# B&R Automation Studio project TestOpenpowerlink
Automation Studio 4.3.11.134 SP

## Configuration Config1

CPU X20CP3586, AutomationRuntime N4.34, Build 4.1.2, Vc V4.34.3

### Task classes (Cpu.sw)
```
Cyclic#4:
  Program <- Program.prg
Libraries: AsIOAcc, runtime, BLLibrarys
```

### Hardware
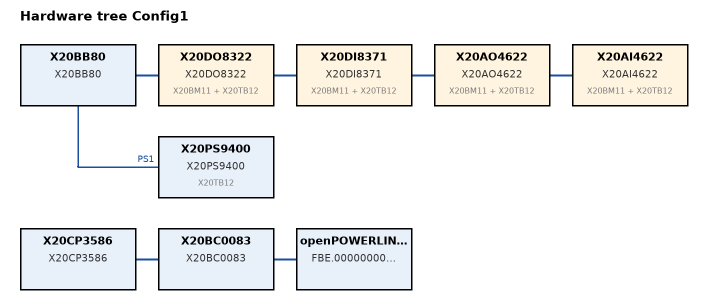
```
X20AI4622 : X20AI4622 v1.0.4.0  [SS1 -> X20TB12d.SS; SL -> X20BM11c.SL1]
  Supervision = off
  LowerLimit = -8192
  ChannelType01 = 4 to 20mA
  ChannelType02 = 4 to 20mA
  ChannelType03 = 4 to 20mA
  ChannelType04 = 4 to 20mA
X20AO4622 : X20AO4622 v1.2.0.0  [SS1 -> X20TB12c.SS; SL -> X20BM11b.SL1]
  Supervision = off
  ChannelType01 = 4 to 20mA
  ChannelType02 = 4 to 20mA
  ChannelType03 = 4 to 20mA
  ChannelType04 = 4 to 20mA
X20BB80 : X20BB80 v1.0.2.0
X20BC0083 : X20BC0083 v2.11.1.0  [PLK1 -> X20CP3586.IF3 (NodeNumber=2) [Cable Type=PowerlinkCable, Length=10, Version=1.0.0.1]; PLK2 -> openPOWERLINK_device.PLK1 (NodeNumber=2) [Cable Type=PowerlinkCable, Length=10, Version=1.0.0.1]; SL -> X20BB80.SL1]
  Supervision = off
X20BM11 : X20BM11 v1.0.0.1  [X2X1 -> X20BB80.IF1]
X20BM11a : X20BM11 v1.0.0.1  [X2X1 -> X20BM11.X2X2]
X20BM11b : X20BM11 v1.0.0.1  [X2X1 -> X20BM11a.X2X2]
X20BM11c : X20BM11 v1.0.0.1  [X2X1 -> X20BM11b.X2X2]
X20CP3586 : X20CP3586 v1.8.1.0
  Connector IF2:
    ActivateDevice = 1
    Mode = Manual
    InternetAddress = 192.168.1.10
    SubnetMask = 255.255.255.0
  Connector IF3:
    CycleTime = 50000
  ConfigurationID = TestOpenpowerlink_Config1
X20DI8371 : X20DI8371 v1.1.0.0  [SS1 -> X20TB12b.SS; SL -> X20BM11a.SL1]
  Supervision = off
X20DO8322 : X20DO8322 v1.3.0.0  [SS1 -> X20TB12a.SS; SL -> X20BM11.SL1]
  Supervision = off
X20PS9400 : X20PS9400 v1.3.0.0  [SS1 -> X20TB12.SS; PS -> X20BB80.PS1]
  Supervision = off
X20TB12 : X20TB12 v1.0.0.0
X20TB12a : X20TB12 v1.0.0.0
X20TB12b : X20TB12 v1.0.0.0
X20TB12c : X20TB12 v1.0.0.0
X20TB12d : X20TB12 v1.0.0.0
openPOWERLINK_device : FBE.00000000_POWERLINK_CiA401_CN (OrderNumber=openPOWERLINK device)  [PLK1 -> X20BC0083.PLK2 (NodeNumber=1) [Cable Type=PowerlinkCable, Length=10, Version=1.0.0.1]]
  Supervision = off
  ResponseTimeout = 2000
  p6000s01_direction = ro
  p6200s01_direction = wo
```

### IoMap.iom - X20CP3586/IoMap.iom
```iecst
VAR_CONFIG
	::Program:array_output[0] AT %QX."X20DO8322".DigitalOutput01;
	::Program:TT001.io.analog_signal AT %IW."X20AI4622".AnalogInput01;
	::Program:TT002.io.analog_signal AT %IW."X20AI4622".AnalogInput02;
	::Program:TT003.io.analog_signal AT %IW."X20AI4622".AnalogInput03;
	::Program:input AT %IB."openPOWERLINK_device".DigitalInput_I6000_S01;
	::Program:output AT %QB."openPOWERLINK_device".DigitalOutput_I6200_S01;
	::Program:module_ok AT %IX."openPOWERLINK_device".ModuleOk;
	::Program:array_output[1] AT %QX."X20DO8322".DigitalOutput02;
	::Program:array_output[2] AT %QX."X20DO8322".DigitalOutput03;
	::Program:array_output[3] AT %QX."X20DO8322".DigitalOutput04;
	::Program:array_output[4] AT %QX."X20DO8322".DigitalOutput05;
	::Program:array_output[5] AT %QX."X20DO8322".DigitalOutput06;
	::Program:array_output[6] AT %QX."X20DO8322".DigitalOutput07;
	::Program:connected AT %QX."X20DO8322".DigitalOutput08;
	::Program:array_input[0] AT %IX."X20DI8371".DigitalInput01;
	::Program:array_input[1] AT %IX."X20DI8371".DigitalInput02;
	::Program:array_input[2] AT %IX."X20DI8371".DigitalInput03;
	::Program:array_input[3]  AT %IX."X20DI8371".DigitalInput04;
	::Program:array_input[4]  AT %IX."X20DI8371".DigitalInput05;
	::Program:array_input[5] AT %IX."X20DI8371".DigitalInput06;
	::Program:array_input[6]  AT %IX."X20DI8371".DigitalInput07;
	::Program:array_input[7]  AT %IX."X20DI8371".DigitalInput08;
END_VAR
```

## Logical view

Binary libraries used (declarations not repeated): operator, runtime, astime, AsIecCon, AsIOAcc


### Program Logical/Program (IEC)

#### Main.st - Init, cyclic, exit code
```iecst
PROGRAM _INIT
	(* Insert code here *)

END_PROGRAM

PROGRAM _CYCLIC
	(* Insert code here *)
	IF clock_ms() - out_delay >= T#1s THEN
		out := NOT out;
		out_delay := clock_ms();
	END_IF;

	array_output[0] := input.0;
	array_output[1] := input.1;
	array_output[2] := input.2;
	array_output[3] := input.3;
	array_output[4] := input.4;
	array_output[5] := input.5;
	array_output[6] := input.6;
	array_output[7] := input.7;

	output.0 := array_input[0];
	output.1 := array_input[1];
	output.2 := array_input[2];
	output.3 := array_input[3];
	output.4 := array_input[4];
	output.5 := array_input[5];
	output.6 := array_input[6];
	output.7 := array_input[7];

	connected := module_ok;

	SensorHandler(TT001, TT001_PARA);
	SensorHandler(TT002, TT002_PARA);
	SensorHandler(TT003, TT003_PARA);

	analog_value := Unscale(value, 100.0, 0.0, SIS_HIGH_LIMIT, SIS_LOW_LIMIT);

	ValveHandler(valve001);
	ValveHandler(valve002);

	RegulatorHandler(regulator001);
	RegulatorHandler(regulator002);

	MotorHandler(motor001);
	MotorHandler(motor002);

	InvertMotorHandler(motor101);
	InvertMotorHandler(motor102);
END_PROGRAM

PROGRAM _EXIT
	(* Insert code here *)

END_PROGRAM
```

#### Variables.var - Local variables
```iecst
VAR
	motor001 : Motor;
	motor102 : InvertMotor;
	motor101 : InvertMotor;
	motor002 : Motor;
	valve002 : Valve;
	valve001 : Valve;
	value : REAL;
	analog_value : INT;
END_VAR
VAR RETAIN
	TT003_PARA : SensorPara;
	TT002_PARA : SensorPara;
	TT001_PARA : SensorPara;
END_VAR
VAR
	TT001 : Sensor;
	out_delay : TIME;
	out : BOOL;
	TT003 : Sensor;
	TT002 : Sensor;
	regulator002 : Regulator;
	regulator001 : Regulator;
	input : USINT;
	output : USINT;
	connected : BOOL;
	module_ok : BOOL;
	array_input : ARRAY[0..7] OF BOOL;
	array_output : ARRAY[0..7] OF BOOL;
END_VAR
```

### Library Logical/BLLibs/BLLibrarys (ANSIC)
Depends on: astime, AsIecCon

#### Types.typ - Exported data types
```iecst
TYPE
	Sensor : 	STRUCT
		io : SensorIO;
		cmd : SensorCmd;
		status : SensorStatus;
		internal : SensorInternal;
	END_STRUCT;
	SensorIO : 	STRUCT
		analog_signal : INT; (*Anolog input*)
	END_STRUCT;
	SensorStatus : 	STRUCT
		value : REAL; (*Process value*)
		gradient_value : REAL; (*ex 1cm / 10s = 0.1 cm/s*)
		state : WORD; (*Bit0: High alarm, Bit1: Low alarm, Bit2: High warnning, Bit3: Low warning, Bit4: High tolerance, Bit5: Low tolerance, Bit6: Gradient alarm, Bit7: Overflow, Bit8: Underflow*)
		high_alarm : BOOL; (*High alarm when the process value upon the set point value -- high_alarm_limit*)
		low_alarm : BOOL; (*Low alarm when the process value under the set point value -- low_alarm_limit*)
		high_warning : BOOL; (*High warning when the process value upon the set point value -- high_warning_limit*)
		low_warning : BOOL; (*Low warning when the process value under the set point value -- low_warning_limit*)
		high_tolerance : BOOL; (*High tolerance when the process value upon the set point value -- high_tolerance_limit*)
		low_tolerance : BOOL; (*Low tolerance when the process value under the set point value -- low_tolerance_limit*)
		gradient_alarm : BOOL; (*Gradient alarm when the absolute value of difference with current value and previous value at last gradient cycle upon the the set value -- gradient_limit*)
		overflow : BOOL; (*The analog signal upon 32767*)
		underflow : BOOL; (*The analog signal under 0-1000*)
	END_STRUCT;
	SensorInternal : 	STRUCT
		high_alarm_timer : TIME; (*Delay timer to output high alarm*)
		low_alarm_timer : TIME; (*Delay timer to output low warning*)
		high_warning_timer : TIME; (*Delay timer to output high alarm*)
		low_warning_timer : TIME; (*Delay timer to output low warning*)
		high_tolerance_timer : TIME; (*Delay timer to output high tolerance*)
		low_tolerance_timer : TIME; (*Delay timer to output low tolerance*)
		gradient_timer : TIME; (*Delay timer to output gradient alarm*)
		pre_value : REAL; (*Record the value at last gradient cycle time*)
		delta_value : REAL; (*Difference of current value and previous value*)
	END_STRUCT;
	SensorCmd : 	STRUCT
		simulation_value : REAL; (*Under simulation mode, the process value will use the simulation value*)
		out_service : BOOL; (*This mode is intended for purposes of maintenance and servicing (replacing the device, for example)*)
		simulation : BOOL; (*This mode is intended for purposes of testing processes or logics (interlock, for example).*)
	END_STRUCT;
	SensorPara : 	STRUCT
		high_range : REAL; (*High scale range for the process value*)
		low_range : REAL; (*Low scale range for the process value*)
		high_alarm_limit : REAL; (*Alarm high*)
		low_alarm_limit : REAL; (*Alarm low*)
		high_warning_limit : REAL; (*Warning high*)
		low_warning_limit : REAL; (*Warning low*)
		high_tolerance_limit : REAL; (*Tolerance high*)
		low_tolerance_limit : REAL; (*Tolerance low*)
		gradient_limit : REAL; (*Positive or negative gradient limit*)
		gradient_cycle : DINT := 10; (*Gradient cycle time*)
		alarm_delay : DINT := 5; (*Alarm delay to outupt *)
		physical_unit : INT; (*Physical unit*)
		high_alarm_enable : BOOL; (*Enable alarm high*)
		low_alarm_enable : BOOL; (*Enable alarm low*)
		high_warning_enable : BOOL; (*Enable warning high*)
		low_warning_enable : BOOL; (*Enable warning low*)
		high_tolerance_enable : BOOL; (*Enable tolerance high*)
		low_tolerance_enable : BOOL; (*Enable tolerance low*)
		gradient_enable : BOOL; (*Enable gradient limit*)
		is_sis : BOOL; (*The analog range value of SIS module is 4000-20000, which is different from normal(0-32767).*)
		inverse : BOOL; (*Inverse the low and high range*)
	END_STRUCT;
	Valve : 	STRUCT
		process : ValveProcess;
		io : ValveIO;
		cmd : ValveCmd;
		status : ValveStatus;
		internal : ValveInternal;
	END_STRUCT;
	ValveProcess : 	STRUCT
		interlock_signal : BOOL;
		auto_open_signal : BOOL;
		stop_signal : BOOL;
		mutex_signal : BOOL;
		open_feedback_state : BOOL;
		close_feedback_state : BOOL;
		error : BOOL;
	END_STRUCT;
	ValveIO : 	STRUCT
		open_feedback : BOOL;
		close_feedback : BOOL;
		valve_open : BOOL;
		emergency_stop : BOOL;
	END_STRUCT;
	ValveStatus : 	STRUCT
		state : WORD; (*Bit0: Open, Bit1: Open feedback, Bit2: Close feedback, Bit3: mutex, Bit4: Open fault, Bit5: Close fault, Bit6: Interlock, Bit7: Emergency stop*)
		mode : BYTE; (*0: Manual mode 1: Automatic mode 2: Local mode 3: Out of service mode*)
		open : BOOL;
		mutex : BOOL;
		interlock : BOOL;
		emergency_stop : BOOL;
		open_fault : BOOL;
		close_fault : BOOL;
		open_feedback : BOOL;
		close_feedback : BOOL;
	END_STRUCT;
	ValveInternal : 	STRUCT
		open_fault_timer : TIME;
		close_fault_timer : TIME;
		manual_open : BOOL;
		mode_edge : BOOL;
	END_STRUCT;
	ValveCmd : 	STRUCT
		open_fault_delay : DINT := 5;
		close_fault_delay : DINT := 5;
		mode : BYTE; (*0: Manual mode 1: Automatic mode 2: Local mode 3: Out of service mode*)
		open : BOOL;
		close : BOOL;
		reset : BOOL;
		open_feedback_enable : BOOL := TRUE;
		close_feedback_enable : BOOL := TRUE;
		mutex_enable : BOOL := TRUE;
		interlock_enable : BOOL := TRUE;
		is_interlock_open : BOOL;
		simulation : BOOL;
	END_STRUCT;
	Regulator : 	STRUCT
		process : RegulatorProcess;
		io : RegulatorIO;
		cmd : RegulatorCmd;
		status : RegulatorStatus;
		internal : RegulatorInternal;
	END_STRUCT;
	RegulatorProcess : 	STRUCT
		auto_position : REAL;
		interlock_signal : BOOL;
		stop_signal : BOOL;
		mutex_signal : BOOL;
		error : BOOL;
	END_STRUCT;
	RegulatorIO : 	STRUCT
		position_feedback : INT;
		position : INT;
		emergency_stop : BOOL;
	END_STRUCT;
	RegulatorStatus : 	STRUCT
		position : REAL;
		position_feedback : REAL;
		state : WORD; (*Bit0: mutex, Bit1: Feedback fault, Bit2: Interlock, Bit3: Emergency stop*)
		mode : BYTE; (*0: Manual mode 1: Automatic mode 2: Local mode 3: Out of service mode*)
		mutex : BOOL;
		interlock : BOOL;
		emergency_stop : BOOL;
		feedback_fault : BOOL;
	END_STRUCT;
	RegulatorInternal : 	STRUCT
		feedback_fault : BOOL;
		feedback_fault_timer : TIME;
	END_STRUCT;
	RegulatorCmd : 	STRUCT
		position : REAL;
		fault_position_delta : REAL := 20.0;
		fault_delay : DINT := 5;
		mode : BYTE; (*0: Manual mode 1: Automatic mode 2: Local mode 3: Out of service mode*)
		reset : BOOL;
		feedback_enable : BOOL := TRUE;
		mutex_enable : BOOL := TRUE;
		interlock_enable : BOOL := TRUE;
		is_interlock_open : BOOL;
		simulation : BOOL;
		inverse : BOOL;
	END_STRUCT;
	Motor : 	STRUCT
		process : MotorProcess;
		io : MotorIO;
		cmd : MotorCmd;
		status : MotorStatus;
		internal : MotorInternal;
	END_STRUCT;
	MotorProcess : 	STRUCT
		run_feedback_state : BOOL;
		stop_feedback_state : BOOL;
		interlock_signal : BOOL;
		auto_run_signal : BOOL;
		stop_signal : BOOL;
		mutex_signal : BOOL;
		error : BOOL;
	END_STRUCT;
	MotorIO : 	STRUCT
		run_feedback : BOOL;
		fault_feedback : BOOL;
		run : BOOL;
		emergency_stop : BOOL;
	END_STRUCT;
	MotorStatus : 	STRUCT
		state : WORD; (*Bit0: Run, Bit1: Run feedback, Bit2: Fault feedback, Bit3: mutex, Bit4: Fault, Bit5: Interlock, Bit6: Emergency stop*)
		mode : BYTE; (*0: Manual mode 1: Automatic mode 2: Local mode 3: Out of service mode*)
		run : BOOL;
		mutex : BOOL;
		interlock : BOOL;
		emergency_stop : BOOL;
		fault : BOOL;
		run_feedback : BOOL;
		fault_feedback : BOOL;
	END_STRUCT;
	MotorInternal : 	STRUCT
		run_fault_timer : TIME;
		jog_timer : TIME;
		jog_run : BOOL;
		manual_run : BOOL;
		mode_edge : BOOL;
	END_STRUCT;
	MotorCmd : 	STRUCT
		fault_delay : DINT := 3;
		jog_delay : DINT := 2;
		mode : BYTE; (*0: Manual mode 1: Automatic mode 2: Local mode 3: Out of service mode*)
		start : BOOL;
		stop : BOOL;
		reset : BOOL;
		jog : BOOL;
		run_feedback_enable : BOOL := TRUE;
		fault_feedback_enable : BOOL := TRUE;
		mutex_enable : BOOL := TRUE;
		interlock_enable : BOOL := TRUE;
		is_interlock_open : BOOL;
		simulation : BOOL;
	END_STRUCT;
	InvertMotor : 	STRUCT
		process : InvertMotorProcess;
		io : InvertMotorIO;
		cmd : InvertMotorCmd;
		status : InvertMotorStatus;
		internal : InvertMotorInternal;
	END_STRUCT;
	InvertMotorProcess : 	STRUCT
		auto_speed : REAL;
		current_feedback : REAL;
		speed_feedback : REAL;
		run_feedback_state : BOOL;
		stop_feedback_state : BOOL;
		interlock_signal : BOOL;
		auto_run_signal : BOOL;
		stop_signal : BOOL;
		mutex_signal : BOOL;
		error : BOOL;
	END_STRUCT;
	InvertMotorIO : 	STRUCT
		run_feedback : BOOL;
		fault_feedback : BOOL;
		run : BOOL;
		emergency_stop : BOOL;
	END_STRUCT;
	InvertMotorStatus : 	STRUCT
		speed : REAL;
		current_feedback : REAL;
		speed_feedback : REAL;
		state : WORD; (*Bit0: Run, Bit1: Run feedback, Bit2: Fault feedback, Bit3: mutex, Bit4: Fault, Bit5: Interlock, Bit6: Emergency stop*)
		mode : BYTE; (*0: Manual mode 1: Automatic mode 2: Local mode 3: Out of service mode*)
		run : BOOL;
		mutex : BOOL;
		interlock : BOOL;
		emergency_stop : BOOL;
		fault : BOOL;
		run_feedback : BOOL;
		fault_feedback : BOOL;
	END_STRUCT;
	InvertMotorInternal : 	STRUCT
		run_fault_timer : TIME;
		jog_timer : TIME;
		jog_run : BOOL;
		manual_run : BOOL;
		mode_edge : BOOL;
	END_STRUCT;
	InvertMotorCmd : 	STRUCT
		speed : REAL;
		fault_delay : DINT := 3;
		jog_delay : DINT := 2;
		mode : BYTE; (*0: Manual mode 1: Automatic mode 2: Local mode 3: Out of service mode*)
		start : BOOL;
		stop : BOOL;
		reset : BOOL;
		jog : BOOL;
		run_feedback_enable : BOOL := TRUE;
		fault_feedback_enable : BOOL := TRUE;
		mutex_enable : BOOL := TRUE;
		interlock_enable : BOOL := TRUE;
		is_interlock_open : BOOL;
		simulation : BOOL;
	END_STRUCT;
END_TYPE
```

#### Constants.var - Exported constants
```iecst
VAR CONSTANT
	DEADBAND_LIMIT : INT := 1000;
	LOW_LIMIT : INT := 0;
	HIGH_LIMIT : INT := 32767;
	SIS_LOW_LIMIT : INT := 4000;
	SIS_HIGH_LIMIT : INT := 20000;
	MANUAL_MODE : BYTE := 0;
	AUTOMATIC_MODE : BYTE := 1;
	LOCAL_MODE : BYTE := 2;
	OUT_SERVICE_MODE : BYTE := 3;
	REGULATOR_POSITION_HIGH : REAL := 100.0;
	REGULATOR_POSITION_LOW : REAL := 0.0;
END_VAR
```

#### BLLibrarys.fun - Exported functions and function blocks
```iecst
{REDUND_OK} FUNCTION SensorHandler : BOOL (*TODO: This is a function that handles sensor*) (*$GROUP=User,$CAT=User,$GROUPICON=User.png,$CATICON=User.png*)
	VAR_INPUT
		sensor : Sensor;
		sensor_para : SensorPara;
	END_VAR
END_FUNCTION

{REDUND_OK} FUNCTION Scale : REAL (*TODO:min-max normalization*) (*$GROUP=User,$CAT=User,$GROUPICON=User.png,$CATICON=User.png*)
	VAR_INPUT
		anolog : INT;
		high_range : REAL;
		low_range : REAL;
		analog_high : INT;
		analog_low : INT;
	END_VAR
END_FUNCTION

{REDUND_OK} FUNCTION Unscale : INT (*TODO: Add your comment here*) (*$GROUP=User,$CAT=User,$GROUPICON=User.png,$CATICON=User.png*)
	VAR_INPUT
		value : REAL;
		high_range : REAL;
		low_range : REAL;
		analog_high : INT;
		analog_low : INT;
	END_VAR
END_FUNCTION

{REDUND_OK} FUNCTION ValveHandler : BOOL (*TODO: Add your comment here*) (*$GROUP=User,$CAT=User,$GROUPICON=User.png,$CATICON=User.png*)
	VAR_INPUT
		valve : Valve;
	END_VAR
END_FUNCTION

{REDUND_OK} FUNCTION OutputDelay : BOOL (*TODO: Delay seconds to output*) (*$GROUP=User,$CAT=User,$GROUPICON=User.png,$CATICON=User.png*)
	VAR_INPUT
		input : BOOL;
		timer : REFERENCE TO TIME;
		second : DINT;
	END_VAR
END_FUNCTION

{REDUND_OK} FUNCTION RegulatorHandler : BOOL (*TODO: Add your comment here*) (*$GROUP=User,$CAT=User,$GROUPICON=User.png,$CATICON=User.png*)
	VAR_INPUT
		regulator : Regulator;
	END_VAR
END_FUNCTION

{REDUND_OK} FUNCTION fabs : REAL (*TODO: Add your comment here*) (*$GROUP=User,$CAT=User,$GROUPICON=User.png,$CATICON=User.png*)
	VAR_INPUT
		value : REAL;
	END_VAR
END_FUNCTION

{REDUND_OK} FUNCTION MotorHandler : BOOL (*TODO: Add your comment here*) (*$GROUP=User,$CAT=User,$GROUPICON=User.png,$CATICON=User.png*)
	VAR_INPUT
		motor : Motor;
	END_VAR
END_FUNCTION

{REDUND_OK} FUNCTION InvertMotorHandler : BOOL (*TODO: Add your comment here*) (*$GROUP=User,$CAT=User,$GROUPICON=User.png,$CATICON=User.png*)
	VAR_INPUT
		motor : InvertMotor;
	END_VAR
END_FUNCTION
```

#### SensorHandler.c
```c
#include <bur/plctypes.h>
#ifdef __cplusplus
	extern "C"
	{
#endif
	#include "BLLibrarys.h"
#ifdef __cplusplus
	};
#endif

/* TODO: This is a function that handles sensor */
plcbit SensorHandler(struct Sensor* sensor, struct SensorPara* sensor_para)
{
	/*Out of service*/
	if (sensor->cmd.out_service)
	{
		sensor->status.overflow = 0;
		sensor->status.underflow = 0;
		sensor->status.value = 0;
		sensor->status.gradient_value = 0;
		sensor->status.high_alarm = 0;
		sensor->status.low_alarm = 0;
		sensor->status.high_warning = 0;
		sensor->status.low_warning = 0;
		sensor->status.high_tolerance = 0;
		sensor->status.low_tolerance = 0;
		sensor->status.gradient_alarm =  0;
		sensor->status.state = 0;
		return 0;
	}

	/*Simulation*/
	if (sensor->cmd.simulation)
	{
		sensor->status.value = sensor->cmd.simulation_value;
	}
	else
	{
		/*Get process value*/
		if(sensor_para->is_sis)
		{
			if(sensor_para->inverse)
				sensor->status.value = Scale(sensor->io.analog_signal, sensor_para->low_range, sensor_para->high_range, SIS_HIGH_LIMIT, SIS_LOW_LIMIT);
			else
				sensor->status.value = Scale(sensor->io.analog_signal, sensor_para->high_range, sensor_para->low_range, SIS_HIGH_LIMIT, SIS_LOW_LIMIT);
		}
		else
		{
			if (sensor_para->inverse)
				sensor->status.value = Scale(sensor->io.analog_signal, sensor_para->low_range, sensor_para->high_range, HIGH_LIMIT, LOW_LIMIT);
			else
				sensor->status.value = Scale(sensor->io.analog_signal, sensor_para->high_range, sensor_para->low_range, HIGH_LIMIT, LOW_LIMIT);
		}
	}

	/*Overflow*/
	sensor->status.overflow = (sensor->io.analog_signal > HIGH_LIMIT)?1:0;

	/*Underflow*/
	sensor->status.underflow = (sensor->io.analog_signal < (LOW_LIMIT - DEADBAND_LIMIT))?1:0;

	/*High alarm*/
	plcbit high_alarm = sensor_para->high_alarm_enable?(sensor->status.value > sensor_para->high_alarm_limit):0;
	sensor->status.high_alarm = OutputDelay(high_alarm, &sensor->process.high_alarm_timer, sensor_para->alarm_delay);

	/*Low alarm*/
	plcbit low_alarm = sensor_para->low_alarm_enable?(sensor->status.value < sensor_para->low_alarm_limit):0;
	sensor->status.low_alarm = OutputDelay(low_alarm, &sensor->process.low_alarm_timer, sensor_para->alarm_delay);

	/*High warning*/
	plcbit high_warning = sensor_para->high_warning_enable?(sensor->status.value > sensor_para->high_warning_limit):0;
	sensor->status.high_warning = OutputDelay(high_warning, &sensor->process.high_warning_timer, sensor_para->alarm_delay);

	/*Low warning*/
	plcbit low_warning = sensor_para->low_warning_enable?(sensor->status.value < sensor_para->low_warning_limit):0;
	sensor->status.low_warning = OutputDelay(low_warning, &sensor->process.low_warning_timer, sensor_para->alarm_delay);

	/*High tolerance*/
	plcbit high_tolerance = sensor_para->high_tolerance_enable?(sensor->status.value > sensor_para->high_tolerance_limit):0;
	sensor->status.high_tolerance = OutputDelay(high_tolerance, &sensor->process.high_tolerance_timer, sensor_para->alarm_delay);

	/*Low tolerance*/
	plcbit low_tolerance = sensor_para->low_tolerance_enable?(sensor->status.value < sensor_para->low_tolerance_limit):0;
	sensor->status.low_tolerance = OutputDelay(low_tolerance, &sensor->process.low_tolerance_timer, sensor_para->alarm_delay);

	/*Gradient alarm*/
	if (sensor_para->gradient_enable)
	{
		if (sensor_para->gradient_cycle <= 0)
		{
			sensor_para->gradient_cycle = 1;
		}
		if ((clock_ms() - sensor->process.gradient_timer) >= (sensor_para->gradient_cycle * 1000))
		{
			float temp = sensor->status.value - sensor->process.pre_value;
			sensor->status.gradient_value = temp / (float)sensor_para->gradient_cycle;
			temp = (temp < 0.0f)?(temp * -1.0f):temp;
			sensor->status.gradient_alarm = (temp > sensor_para->gradient_limit)?1:0;
			sensor->process.pre_value = sensor->status.value;
			sensor->process.gradient_timer = clock_ms();
		}
	}
	else
	{
		sensor->status.gradient_alarm = 0;
	}

	sensor->status.state = (sensor->status.high_alarm | (sensor->status.low_alarm << 1) | (sensor->status.high_warning << 2)  | (sensor->status.low_warning << 3) |
		(sensor->status.high_tolerance << 4) | (sensor->status.low_tolerance << 5)  | (sensor->status.gradient_alarm << 6)  | (sensor->status.overflow << 7) | (sensor->status.underflow << 8));

	return 1;
}
```

#### Scale.c
```c
#include <bur/plctypes.h>
#ifdef __cplusplus
	extern "C"
	{
#endif
	#include "BLLibrarys.h"
#ifdef __cplusplus
	};
#endif
/* TODO:min-max normalization */
float Scale(signed short analog, float high_range, float low_range, signed short analog_high, signed short analog_low)
{
	/*TODO: Add your code here*/
	float temp;
	if (analog < analog_low)
	{
		return low_range;
	}

	if (analog > analog_high)
	{
		return high_range;
	}

	temp = (float)(analog - analog_low) * (high_range - low_range) / (float)(analog_high - analog_low) + low_range;
	return temp;
}
```

#### Unscale.c
```c
#include <bur/plctypes.h>
#ifdef __cplusplus
	extern "C"
	{
#endif
	#include "BLLibrarys.h"
#ifdef __cplusplus
	};
#endif
/* TODO: Add your comment here */
signed short Unscale(float value, float high_range, float low_range, signed short analog_high, signed short analog_low)
{
	/*TODO: Add your code here*/
	if(high_range == low_range)
	{
		return analog_low;
	}

	if (value < low_range)
	{
		return analog_low;
	}

	if (value > high_range)
	{
		return analog_high;
	}

	return ((signed short)(value - low_range) * (analog_high - analog_low) / (signed short)(high_range - low_range) + analog_low);
}
```

#### ValveHandler.c
```c
#include <bur/plctypes.h>
#ifdef __cplusplus
	extern "C"
	{
#endif
	#include "BLLibrarys.h"
#ifdef __cplusplus
	};
#endif
/* TODO: Add your comment here */
plcbit ValveHandler(struct Valve* valve)
{
	/*TODO: Add your code here*/
	/* Mode select*/
	valve->status.mode = valve->cmd.mode;

	/*Out of service mode*/
	if (valve->status.mode == OUT_SERVICE_MODE)
	{
		valve->status.open_fault = 0;
		valve->status.close_fault = 0;
		valve->status.emergency_stop = 0;
		valve->status.interlock = 0;
		valve->status.mutex = 0;
		valve->status.open = 0;
		valve->status.open_feedback = 0;
		valve->status.close_feedback = 0;
		valve->status.state = 0;
		return 0;
	}

	/*Local mode*/
	if(valve->status.mode == LOCAL_MODE)
	{
		valve->status.open = valve->io.open_feedback;
		valve->status.open_feedback = valve->io.open_feedback;
		valve->status.close_feedback = valve->io.close_feedback;
		valve->status.emergency_stop = valve->io.emergency_stop;
		valve->status.interlock = 0;
		valve->status.mutex = 0;
		valve->status.open_fault = 0;
		valve->status.close_fault = 0;
		valve->status.state = valve->status.open | (valve->status.open_feedback << 1) | (valve->status.close_feedback << 2) | (valve->status.emergency_stop << 3) |
			(valve->status.interlock << 4) | (valve->status.mutex << 5) | (valve->status.open_fault << 6) | (valve->status.close_fault << 7);
		return 1;
	}

	/**/
	if (valve->para.open_feedback_enable && valve->para.close_feedback_enable)
	{
		valve->input.open_feedback_state = valve->status.open && valve->io.open_feedback && !valve->io.close_feedback;
		valve->input.close_feedback_state = !valve->status.open && !valve->io.open_feedback && valve->io.close_feedback;
	}
	else if(valve->para.open_feedback_enable && !valve->para.close_feedback_enable)
	{
		valve->input.open_feedback_state = valve->status.open && valve->io.open_feedback;
		valve->input.close_feedback_state = !valve->status.open && !valve->io.open_feedback;
	}
	else if (!valve->para.open_feedback_enable && valve->para.close_feedback_enable)
	{
		valve->input.open_feedback_state = valve->status.open && !valve->io.close_feedback;
		valve->input.close_feedback_state = !valve->status.open && valve->io.close_feedback;
	}
	else
	{
		valve->input.open_feedback_state = valve->status.open;
		valve->input.close_feedback_state = !valve->status.open;
	}

	/*Emergency stop*/
	if (valve->io.emergency_stop | valve->input.stop_signal)
	{
		valve->status.emergency_stop = 1;
	}
	else
	{
		if(valve->cmd.reset)
		{
			valve->status.emergency_stop = 0;
		}
	}

	/*Interlock*/
	if (valve->input.interlock_signal)
	{
		valve->status.interlock = 1;
	}
	else
	{
		if(valve->cmd.reset)
		{
			valve->status.interlock = 0;
		}
	}

	/*Mutex*/
	valve->status.mutex = valve->input.mutex_signal && !valve->cmd.mutex_disable;

	/*Feedback state*/
	valve->status.open_feedback = valve->io.open_feedback;
	valve->status.close_feedback = valve->io.close_feedback;

	/*Feedback fault*/
	valve->status.open_fault = OutputDelay((valve->status.open && !valve->input.open_feedback_state), &valve->process.open_fault_timer, valve->para.open_fault_delay);
	valve->status.close_fault = OutputDelay((!valve->status.open && !valve->input.close_feedback_state), &valve->process.close_fault_timer, valve->para.close_fault_delay);

	/*Automatic mode*/
	if(valve->status.mode == AUTOMATIC_MODE)
	{
		if (valve->para.is_interlock_open)
		{
			valve->status.open = valve->status.interlock || (valve->input.auto_open_signal && !valve->status.emergency_stop && !valve->status.mutex);
		}
		else
		{
			valve->status.open = valve->input.auto_open_signal && !valve->status.emergency_stop && !valve->status.interlock && !valve->status.mutex;
		}
	}

	/*Manual mode*/
	if (valve->status.mode == MANUAL_MODE)
	{
		if (valve->para.is_interlock_open)
		{
			plcbit manual_open;

			if (valve->cmd.open && !valve->status.emergency_stop && !valve->status.mutex)
			{
				manual_open = 1;
			}
			if (valve->cmd.close || valve->status.emergency_stop || valve->status.mutex)
			{
				manual_open = 0;
			}
			valve->status.open = valve->status.interlock || manual_open;
		}
		else
		{
			if (valve->cmd.open && !valve->status.emergency_stop && !valve->status.interlock && !valve->status.mutex)
			{
				valve->status.open = 1;
			}
			if (valve->cmd.close || valve->status.emergency_stop || valve->status.interlock || valve->status.mutex)
			{
				valve->status.open = 0;
			}
		}
	}

	/*Output*/
	valve->io.valve_open = valve->status.open;

	/*Reset command*/
	if (valve->cmd.open)
	{
		valve->cmd.open = 0;
	}
	if (valve->cmd.close)
	{
		valve->cmd.close = 0;
	}
	if (valve->cmd.reset)
	{
		valve->cmd.reset = 0;
	}

	return 1;
}
```

#### OutputDelay.c
```c
#include <bur/plctypes.h>
#ifdef __cplusplus
	extern "C"
	{
#endif
	#include "BLLibrarys.h"
#ifdef __cplusplus
	};
#endif
/* TODO: Delay seconds to output */
plcbit OutputDelay(plcbit input, plctime* timer, signed long second)
{
	/*TODO: Add your code here*/
	plcbit output = 0;
	if(input)
	{
		if((clock_ms() - *timer) >= (second * 1000))
		{
			output = 1;
		}
	}
	else
	{
		output = 0;
		*timer = clock_ms();
	}
	return output;
}
```

#### RegulatorHandler.c
```c
#include <bur/plctypes.h>
#ifdef __cplusplus
	extern "C"
	{
#endif
#include "BLLibrarys.h"
#ifdef __cplusplus
	};
#endif

#define FAULT_BITS 0xFFFC

static void reset_cmd(struct RegulatorCmd* cmd);

/* TODO: Add your comment here */
plcbit RegulatorHandler(struct Regulator* regulator)
{
	/*TODO: Add your code here*/
	/* Mode select*/
	regulator->status.mode = regulator->cmd.mode;

	/*Out of service mode*/
	if (regulator->status.mode == OUT_SERVICE_MODE)
	{
		regulator->status.position = 0.0f;
		regulator->status.position_feedback = 0.0f;
		regulator->status.feedback_fault = 0;
		regulator->status.emergency_stop = 0;
		regulator->status.interlock = 0;
		regulator->status.mutex = 0;
		regulator->status.state = 0;
		reset_cmd(&(regulator->cmd));
		return 0;
	}

	/*Local mode*/
	if(regulator->status.mode == LOCAL_MODE)
	{
		if (regulator->cmd.inverse)
		{
			regulator->status.position_feedback = Scale(regulator->io.position_feedback, REGULATOR_POSITION_LOW, REGULATOR_POSITION_HIGH, HIGH_LIMIT, LOW_LIMIT);
		}
		else
		{
			regulator->status.position_feedback = Scale(regulator->io.position_feedback, REGULATOR_POSITION_HIGH, REGULATOR_POSITION_LOW, HIGH_LIMIT, LOW_LIMIT);
		}
		regulator->status.position = regulator->status.position_feedback;
		regulator->status.emergency_stop = regulator->io.emergency_stop;
		regulator->status.interlock = 0;
		regulator->status.mutex = 0;
		regulator->status.feedback_fault = 0;
		regulator->status.state = regulator->status.mutex | (regulator->status.feedback_fault << 1) | (regulator->status.interlock << 2) | (regulator->status.emergency_stop << 3);
		reset_cmd(&(regulator->cmd));
		return 1;
	}

	/*Simulation*/
	if (regulator->cmd.simulation)
	{
		regulator->status.position_feedback = regulator->status.position;
	}
	else
	{
		if (regulator->cmd.feedback_enable)
		{
			/*Feedback position*/
			if (regulator->cmd.inverse)
			{
				regulator->status.position_feedback = Scale(regulator->io.position_feedback, REGULATOR_POSITION_LOW, REGULATOR_POSITION_HIGH, HIGH_LIMIT, LOW_LIMIT);
			}
			else
			{
				regulator->status.position_feedback = Scale(regulator->io.position_feedback, REGULATOR_POSITION_HIGH, REGULATOR_POSITION_LOW, HIGH_LIMIT, LOW_LIMIT);
			}
		}
		else
		{
			/*Feedback position*/
			regulator->status.position_feedback = 0.0f;
		}
	}

	/*Emergency stop*/
	if (regulator->io.emergency_stop | regulator->process.stop_signal)
	{
		regulator->status.emergency_stop = 1;
	}
	else
	{
		if(regulator->cmd.reset)
		{
			regulator->status.emergency_stop = 0;
		}
	}

	/*Interlock*/
	if (regulator->cmd.interlock_enable)
	{
		if (regulator->process.interlock_signal)
		{
			regulator->status.interlock = 1;
		}
		else
		{
			if(regulator->cmd.reset)
			{
				regulator->status.interlock = 0;
			}
		}
	}
	else
	{
		regulator->status.interlock = 0;
	}

	/*Mutex*/
	regulator->status.mutex = regulator->process.mutex_signal && regulator->cmd.mutex_enable;

	/*Feedback fault*/
	if (regulator->cmd.feedback_enable)
	{
		if (fabs(regulator->status.position - regulator->status.position_feedback) > regulator->cmd.fault_position_delta)
		{
			regulator->internal.feedback_fault = 1;
		}
		else
		{
			regulator->internal.feedback_fault = 0;
		}
	}
	else
	{
		regulator->internal.feedback_fault = 0;
	}
	regulator->status.feedback_fault = OutputDelay(regulator->internal.feedback_fault, &regulator->internal.feedback_fault_timer, regulator->cmd.fault_delay);

	/*Automatic mode*/
	if(regulator->status.mode == AUTOMATIC_MODE)
	{
		if (regulator->cmd.is_interlock_open)
		{
			if (regulator->status.interlock)
			{
				regulator->status.position = 100.0f;
			}
			else
			{
				if ((!regulator->status.emergency_stop) && (!regulator->status.mutex))
				{
					regulator->status.position = regulator->process.auto_position;
				}
				else
				{
					regulator->status.position = 0.0f;
				}
			}
		}
		else
		{
			if ((!regulator->status.emergency_stop) && (!regulator->status.interlock) && (!regulator->status.mutex))
			{
				regulator->status.position = regulator->process.auto_position;
			}
			else
			{
				regulator->status.position = 0.0f;
			}
		}
	}

	/*Manual mode*/
	if (regulator->status.mode == MANUAL_MODE)
	{
		if (regulator->cmd.is_interlock_open)
		{
			if (regulator->status.interlock)
			{
				regulator->status.position = 100.0f;
			}
			else
			{
				if ((!regulator->status.emergency_stop) && (!regulator->status.mutex))
				{
					regulator->status.position = regulator->cmd.position;
				}
				else
				{
					regulator->status.position = 0.0f;
				}
			}
		}
		else
		{
			if ((!regulator->status.emergency_stop) && (!regulator->status.interlock) && (!regulator->status.mutex))
			{
				regulator->status.position = regulator->cmd.position;
			}
			else
			{
				regulator->status.position = 0.0f;
			}
		}
	}

	regulator->status.state = regulator->status.mutex | (regulator->status.feedback_fault << 1) | (regulator->status.interlock << 2) | (regulator->status.emergency_stop << 3);
	regulator->process.error = (regulator->status.state & FAULT_BITS)?1:0;

	/*Reset command*/
	reset_cmd(&(regulator->cmd));

	/*Output*/
	if (regulator->cmd.simulation)
	{
		regulator->io.position = 0;
	}
	else
	{
		if (regulator->cmd.inverse)
		{
			regulator->io.position = Unscale(regulator->status.position, REGULATOR_POSITION_HIGH, REGULATOR_POSITION_LOW, LOW_LIMIT, HIGH_LIMIT);
		}
		else
		{
			regulator->io.position = Unscale(regulator->status.position, REGULATOR_POSITION_HIGH, REGULATOR_POSITION_LOW, HIGH_LIMIT, LOW_LIMIT);
		}
	}

	return 1;
}

	/*Reset command*/
static void reset_cmd(struct RegulatorCmd* cmd)
{
	if (cmd->reset)
	{
		cmd->reset = 0;
	}
}
```

#### fabs.c
```c
#include <bur/plctypes.h>
#ifdef __cplusplus
	extern "C"
	{
#endif
	#include "BLLibrarys.h"
#ifdef __cplusplus
	};
#endif
/* TODO: Add your comment here */
float fabs(float value)
{
	/*TODO: Add your code here*/
	if (value < 0.0f)
	{
		return -(value);
	}
	else
	{
		return (value);
	}
}
```

#### MotorHandler.c
```c
#include <bur/plctypes.h>
#ifdef __cplusplus
	extern "C"
	{
#endif
#include "BLLibrarys.h"
#ifdef __cplusplus
	};
#endif

#define FAULT_BITS 0xFFF0

static void reset_cmd(struct MotorCmd* cmd);

/* TODO: Add your comment here */
plcbit MotorHandler(struct Motor* motor)
{
	/*TODO: Add your code here*/
	/* Mode select*/
	motor->status.mode = motor->cmd.mode;

	/*Out of service mode*/
	if (motor->status.mode == OUT_SERVICE_MODE)
	{
		motor->internal.mode_edge = 0;
		motor->status.fault = 0;
		motor->status.emergency_stop = 0;
		motor->status.interlock = 0;
		motor->status.mutex = 0;
		motor->status.run = 0;
		motor->status.run_feedback = 0;
		motor->status.fault_feedback = 0;
		motor->status.state = 0;
		reset_cmd(&(motor->cmd));
		return 0;
	}

	/*Local mode*/
	if(motor->status.mode == LOCAL_MODE)
	{
		motor->internal.mode_edge = 0;
		motor->status.run = motor->io.run_feedback;
		motor->status.run_feedback = motor->io.run_feedback;
		motor->status.fault_feedback = motor->io.fault_feedback;
		motor->status.emergency_stop = motor->io.emergency_stop;
		motor->status.interlock = 0;
		motor->status.mutex = 0;
		motor->status.fault = motor->io.fault_feedback;
		motor->status.state = motor->status.run | (motor->status.run_feedback << 1) | (motor->status.fault_feedback << 2) | (motor->status.mutex << 3) |
			(motor->status.fault << 4) | (motor->status.interlock << 5) | (motor->status.emergency_stop << 6);
		reset_cmd(&(motor->cmd));
		return 1;
	}

	/*Simulation*/
	if (motor->cmd.simulation)
	{
		motor->process.run_feedback_state = motor->status.run;
		motor->process.stop_feedback_state = !motor->status.run;
	}
	else
	{
		if (motor->cmd.run_feedback_enable && motor->cmd.fault_feedback_enable)
		{
			motor->process.run_feedback_state = motor->status.run && motor->io.run_feedback && !motor->io.fault_feedback;
			motor->process.stop_feedback_state = !motor->status.run && !motor->io.run_feedback && !motor->io.fault_feedback;
		}
		else if(motor->cmd.run_feedback_enable && !motor->cmd.fault_feedback_enable)
		{
			motor->process.run_feedback_state = motor->status.run && motor->io.run_feedback;
			motor->process.stop_feedback_state = !motor->status.run && !motor->io.run_feedback;

		}
		else if (!motor->cmd.run_feedback_enable && motor->cmd.fault_feedback_enable)
		{
			motor->process.run_feedback_state = motor->status.run && !motor->io.fault_feedback;
			motor->process.stop_feedback_state = !motor->status.run && !motor->io.fault_feedback;
		}
		else
		{
			motor->process.run_feedback_state = motor->status.run;
			motor->process.stop_feedback_state = !motor->status.run;
		}
	}

	/*Emergency stop*/
	if (motor->io.emergency_stop | motor->process.stop_signal)
	{
		motor->status.emergency_stop = 1;
	}
	else
	{
		if(motor->cmd.reset)
		{
			motor->status.emergency_stop = 0;
		}
	}

	/*Interlock*/
	if (motor->cmd.interlock_enable)
	{
		if (motor->process.interlock_signal)
		{
			motor->status.interlock = 1;
		}
		else
		{
			if(motor->cmd.reset)
			{
				motor->status.interlock = 0;
			}
		}
	}
	else
	{
		motor->status.interlock = 0;
	}

	/*Mutex*/
	motor->status.mutex = motor->process.mutex_signal && motor->cmd.mutex_enable;

	/*Feedback state*/
	motor->status.run_feedback = motor->io.run_feedback;
	motor->status.fault_feedback = motor->io.fault_feedback;

	/*Feedback fault*/
	if (OutputDelay((motor->status.run && !motor->process.run_feedback_state) || (!motor->status.run && !motor->process.stop_feedback_state), &motor->internal.run_fault_timer, motor->cmd.fault_delay))
	{
		motor->status.fault = 1;
	}
	else
	{
		if(motor->cmd.reset)
		{
			motor->status.fault = 0;
		}
	}

	/*Automatic mode*/
	if(motor->status.mode == AUTOMATIC_MODE)
	{
		motor->internal.mode_edge = 0;
		if (motor->cmd.is_interlock_open)
		{
			motor->status.run = motor->status.interlock || (motor->process.auto_run_signal && !motor->status.fault && !motor->status.emergency_stop && !motor->status.mutex);
		}
		else
		{
			motor->status.run = motor->process.auto_run_signal && !motor->status.fault && !motor->status.emergency_stop && !motor->status.interlock && !motor->status.mutex;
		}
	}

	/*Manual mode*/
	if (motor->status.mode == MANUAL_MODE && !motor->internal.mode_edge)
	{
		/*Reset open state, when the mode switch from others to manual*/
		motor->status.run = 0;
		motor->internal.mode_edge = 1;
	}
	if (motor->status.mode == MANUAL_MODE)
	{
		if (motor->cmd.jog && !motor->status.fault && !motor->status.emergency_stop && !motor->status.interlock && !motor->status.mutex)
			{
			motor->internal.jog_run = 1;
		}
		if(motor->internal.jog_run)
		{
			if((clock_ms() - motor->internal.jog_timer) >= (motor->cmd.jog_delay * 1000))
			{
				motor->internal.jog_run = 0;
			}
		}
		else
		{
			motor->internal.jog_timer = clock_ms();
		}

		if (motor->cmd.is_interlock_open)
		{
			if (motor->cmd.start && !motor->status.fault && !motor->status.emergency_stop && !motor->status.mutex)
			{
				motor->internal.manual_run = 1;
			}
			if (motor->cmd.stop || motor->status.fault || motor->status.emergency_stop || motor->status.mutex)
			{
				motor->internal.manual_run = 0;
			}
			motor->status.run = motor->status.interlock || motor->status.fault || motor->internal.manual_run || motor->internal.jog_run;
		}
		else
		{
			if (motor->cmd.start && !motor->status.fault && !motor->status.emergency_stop && !motor->status.interlock && !motor->status.mutex)
			{
				motor->internal.manual_run = 1;
			}
			if (motor->cmd.stop || motor->status.fault || motor->status.emergency_stop || motor->status.interlock || motor->status.mutex)
			{
				motor->internal.manual_run = 0;
			}
			motor->status.run = motor->internal.manual_run || motor->internal.jog_run;
		}
	}

	motor->status.state = motor->status.run | (motor->status.run_feedback << 1) | (motor->status.fault_feedback << 2) | (motor->status.mutex << 3) |
		(motor->status.fault << 4) | (motor->status.interlock << 5) | (motor->status.emergency_stop << 6);

	motor->process.error = (motor->status.state & FAULT_BITS)?1:0;

	/*Reset command*/
	reset_cmd(&(motor->cmd));

	/*Output*/
	if (motor->cmd.simulation)
	{
		motor->io.run = 0;
	}
	else
	{
		motor->io.run = motor->status.run;
	}

	return 1;
}

/*Reset command*/
static void reset_cmd(struct MotorCmd* cmd)
{
	if (cmd->start)
	{
		cmd->start = 0;
	}
	if (cmd->stop)
	{
		cmd->stop = 0;
	}
	if (cmd->jog)
	{
		cmd->jog = 0;
	}
	if (cmd->reset)
	{
		cmd->reset = 0;
	}
}
```

#### InvertMotorHandler.c
```c
#include <bur/plctypes.h>
#ifdef __cplusplus
	extern "C"
	{
#endif
	#include "BLLibrarys.h"
#ifdef __cplusplus
	};
#endif

#define FAULT_BITS 0xFFF0

static void reset_cmd(struct InvertMotorCmd* cmd);

/* TODO: Add your comment here */
plcbit InvertMotorHandler(struct InvertMotor* motor)
{
	/*TODO: Add your code here*/
	/* Mode select*/
	motor->status.mode = motor->cmd.mode;

	/*Out of service mode*/
	if (motor->status.mode == OUT_SERVICE_MODE)
	{
		motor->internal.mode_edge = 0;
		motor->status.fault = 0;
		motor->status.emergency_stop = 0;
		motor->status.interlock = 0;
		motor->status.mutex = 0;
		motor->status.run = 0;
		motor->status.run_feedback = 0;
		motor->status.fault_feedback = 0;
		motor->status.state = 0;
		motor->status.current_feedback = 0;
		motor->status.speed_feedback = 0;
		motor->status.speed = 0;
		reset_cmd(&(motor->cmd));
		return 0;
	}

	/*Local mode*/
	if(motor->status.mode == LOCAL_MODE)
	{
		motor->internal.mode_edge = 0;
		motor->status.run = motor->io.run_feedback;
		motor->status.run_feedback = motor->io.run_feedback;
		motor->status.fault_feedback = motor->io.fault_feedback;
		motor->status.emergency_stop = motor->io.emergency_stop;
		motor->status.interlock = 0;
		motor->status.mutex = 0;
		motor->status.fault = motor->io.fault_feedback;
		motor->status.current_feedback = motor->process.current_feedback;
		motor->status.speed_feedback = motor->process.speed_feedback;
		motor->status.speed = 0;
		motor->status.state = motor->status.run | (motor->status.run_feedback << 1) | (motor->status.fault_feedback << 2) | (motor->status.mutex << 3) |
			(motor->status.fault << 4) | (motor->status.interlock << 5) | (motor->status.emergency_stop << 6);
		reset_cmd(&(motor->cmd));
		return 1;
	}

	/*Simulation*/
	if (motor->cmd.simulation)
	{
		motor->process.run_feedback_state = motor->status.run;
		motor->process.stop_feedback_state = !motor->status.run;
	}
	else
	{
		if (motor->cmd.run_feedback_enable && motor->cmd.fault_feedback_enable)
		{
			motor->process.run_feedback_state = motor->status.run && motor->io.run_feedback && !motor->io.fault_feedback;
			motor->process.stop_feedback_state = !motor->status.run && !motor->io.run_feedback && !motor->io.fault_feedback;
		}
		else if(motor->cmd.run_feedback_enable && !motor->cmd.fault_feedback_enable)
		{
			motor->process.run_feedback_state = motor->status.run && motor->io.run_feedback;
			motor->process.stop_feedback_state = !motor->status.run && !motor->io.run_feedback;

		}
		else if (!motor->cmd.run_feedback_enable && motor->cmd.fault_feedback_enable)
		{
			motor->process.run_feedback_state = motor->status.run && !motor->io.fault_feedback;
			motor->process.stop_feedback_state = !motor->status.run && !motor->io.fault_feedback;
		}
		else
		{
			motor->process.run_feedback_state = motor->status.run;
			motor->process.stop_feedback_state = !motor->status.run;
		}
	}

	/*Emergency stop*/
	if (motor->io.emergency_stop | motor->process.stop_signal)
	{
		motor->status.emergency_stop = 1;
	}
	else
	{
		if(motor->cmd.reset)
		{
			motor->status.emergency_stop = 0;
		}
	}

	/*Interlock*/
	if (motor->cmd.interlock_enable)
	{
		if (motor->process.interlock_signal)
		{
			motor->status.interlock = 1;
		}
		else
		{
			if(motor->cmd.reset)
			{
				motor->status.interlock = 0;
			}
		}
	}
	else
	{
		motor->status.interlock = 0;
	}

	/*Mutex*/
	motor->status.mutex = motor->process.mutex_signal && motor->cmd.mutex_enable;

	/*Feedback state*/
	motor->status.current_feedback = motor->process.current_feedback;
	motor->status.speed_feedback = motor->process.speed_feedback;
	motor->status.run_feedback = motor->io.run_feedback;
	motor->status.fault_feedback = motor->io.fault_feedback;

	/*Feedback fault*/
	if (OutputDelay((motor->status.run && !motor->process.run_feedback_state) || (!motor->status.run && !motor->process.stop_feedback_state), &motor->internal.run_fault_timer, motor->cmd.fault_delay))
	{
		motor->status.fault = 1;
	}
	else
	{
		if(motor->cmd.reset)
		{
			motor->status.fault = 0;
		}
	}

	/*Automatic mode*/
	if(motor->status.mode == AUTOMATIC_MODE)
	{
		motor->internal.mode_edge = 0;

		motor->status.speed = motor->process.auto_speed;

		if (motor->cmd.is_interlock_open)
		{
			motor->status.run = motor->status.interlock || (motor->process.auto_run_signal && !motor->status.fault && !motor->status.emergency_stop && !motor->status.mutex);
		}
		else
		{
			motor->status.run = motor->process.auto_run_signal && !motor->status.fault && !motor->status.emergency_stop && !motor->status.interlock && !motor->status.mutex;
		}
	}

	/*Manual mode*/
	if (motor->status.mode == MANUAL_MODE && !motor->internal.mode_edge)
	{
		/*Reset open state, when the mode switch from others to manual*/
		motor->status.run = 0;
		motor->internal.mode_edge = 1;
	}
	if (motor->status.mode == MANUAL_MODE)
	{
		motor->status.speed = motor->cmd.speed;

		if (motor->cmd.jog && !motor->status.fault && !motor->status.emergency_stop && !motor->status.interlock && !motor->status.mutex)
		{
			motor->internal.jog_run = 1;
		}
		if(motor->internal.jog_run)
		{
			if((clock_ms() - motor->internal.jog_timer) >= (motor->cmd.jog_delay * 1000))
			{
				motor->internal.jog_run = 0;
			}
		}
		else
		{
			motor->internal.jog_timer = clock_ms();
		}

		if (motor->cmd.is_interlock_open)
		{
			if (motor->cmd.start && !motor->status.fault && !motor->status.emergency_stop && !motor->status.mutex)
			{
				motor->internal.manual_run = 1;
			}
			if (motor->cmd.stop || motor->status.fault || motor->status.emergency_stop || motor->status.mutex)
			{
				motor->internal.manual_run = 0;
			}
			motor->status.run = motor->status.interlock || motor->status.fault || motor->internal.manual_run || motor->internal.jog_run;
		}
		else
		{
			if (motor->cmd.start && !motor->status.fault && !motor->status.emergency_stop && !motor->status.interlock && !motor->status.mutex)
			{
				motor->internal.manual_run = 1;
			}
			if (motor->cmd.stop || motor->status.fault || motor->status.emergency_stop || motor->status.interlock || motor->status.mutex)
			{
				motor->internal.manual_run = 0;
			}
			motor->status.run = motor->internal.manual_run || motor->internal.jog_run;
		}
	}

	motor->status.state = motor->status.run | (motor->status.run_feedback << 1) | (motor->status.fault_feedback << 2) | (motor->status.mutex << 3) |
		(motor->status.fault << 4) | (motor->status.interlock << 5) | (motor->status.emergency_stop << 6);

	motor->process.error = (motor->status.state & FAULT_BITS)?1:0;

	/*Reset command*/
	reset_cmd(&(motor->cmd));

	/*Output*/
	if (motor->cmd.simulation)
	{
		motor->io.run = 0;
	}
	else
	{
		motor->io.run = motor->status.run;
	}

	return 1;
}

/*Reset command*/
static void reset_cmd(struct InvertMotorCmd* cmd)
{
	if (cmd->start)
	{
		cmd->start = 0;
	}
	if (cmd->stop)
	{
		cmd->stop = 0;
	}
	if (cmd->jog)
	{
		cmd->jog = 0;
	}
	if (cmd->reset)
	{
		cmd->reset = 0;
	}
}
```

Listed in the project but not available here: Logical/Global.typ, Logical/Global.var, Logical/Program/Types.typ
